Fanuc KAREL source: IO0015.KL

-- PROVISIONAL review KL for V940-1; original PC SHA256 abff448b500ceff28b4b85445393b7a4ca6b36391ff79d0e0dffb7653b4b237a
-- Incomplete behavior may be omitted. Consult companion uncertainty JSON. Do not deploy.
PROGRAM IO0015
%NOLOCKGROUP
-- UNRESOLVED_LOCAL_POOL 5 cells at code offset 13; source declarations unknown
-- DIRECT_LOCAL_WORD_ACCESS alone does not prove INTEGER, REAL, or BOOLEAN
BEGIN
  -- V9_ZERO_TABLE_METADATA_HINT layout=0001; no indexed target words; source/name/runtime held
  -- V9_ZERO_GLOBAL_LAYOUT_HINT count-one $GROUP table, zero relocation slots, two routine descriptors; executable preamble and source held
  -- UNRESOLVED_PC offsets 0-18; opcodes 2B,2C,7B
  -- UNRESOLVED_PC offsets 23-30; opcodes 9D,23
  -- UNRESOLVED_PC offsets 35-49; opcodes 2E,22,9D,33,35
  -- UNRESOLVED_PC offsets 54-61; opcodes 9D,23
  -- UNRESOLVED_PC offsets 66-77; opcodes 2E,23
  -- UNRESOLVED_PC offsets 82-106; opcodes 03,22,21,33,34,1B,9D,12,13,04,14
  -- UNRESOLVED_PC offsets 111-115; opcodes 7F
  -- UNRESOLVED_PC offsets 120-124; opcodes 27,AA
  -- UNRESOLVED_PC offsets 129-133; opcodes 7F
END IO0015
